PROGRAM Main
VAR
	// JaWa
	_iDbg:INT;	
	_download5:BOOL;
	//Enum1: FanControlTypes := FanControlTypes.Flow;
	GreenMaster: GreenMasterXXL_FB;
	StartupDone: BOOL;
	EventLog: EventLog;
	xxx: bool;
	Saver: FB_S_UPS_CX81xx;
	HostName: FB_GetHostName;
	UseReverse_C_QN1: BOOL;
	test1: bool;
	
	Std_Interface : Standard_Interface;
	CTH_Interface: CTH_Interface;
	Stena_Interface: Stena_Interface;
	ExtraAlarms_Interface: ExtraAlarms_Interface;
	SmokeControl_Interface: SmokeControl_Interface;

	Redundancy:Redundancy;
	ParallelUnits: ParallelUnits;
	
	GreenMasterDI: GreenMasterDI;
	GreenMasterDO: GreenMasterDO;
	GreenMasterAI: GreenMasterAI;
	GreenMasterAO: GreenMasterAO;
	GreenMasterAI2_RTU: GreenMasterAIU_ModbusRTU;
	AnySensorError: BOOL;
	{attribute 'TcEncoding':='UTF-8'}
	str: STRING;
	n: INT;
	
	NightCooling: BOOL;
	DebugStop: BOOL;
	WritePersistentData: WritePersistentData;
	StartWritePersistentData: BOOL;
	SavedParameters: GreenMasterBaseParameters;
	DevMon: DeviationMonitor;
	DevValue: LREAL;
	TestPID: TestPID;
	fbTime : FB_LocalSystemTime := ( bEnable := TRUE, dwCycle := 1 );
	LastSecondsCounter: LINT;
    sTime: STRING;	
	sPart1: STRING;
	sPart2: STRING;
	ExceptionYet: BOOL;
	PTest: POINTER TO BYTE;
	Crash: BOOL;
	i: INT;
	w: WORD;
	Rr: LREAL;
END_VAR
VAR PERSISTENT
END_VAR

IF NOT ExceptionYet THEN
	__TRY
		EventLog(EventLogData := Globals.EventLog);
		IF NOT StartupDone THEN
			Globals.SystemStartTime := NowDT();
			EventLog.LogEvent(Message := 'Starting up', Kind := EventTypes.Information);
			//EventLog.LogEventJSON(Message := 'Test data $${KFactor} and $${PressureControl.SP}', Kind := EventTypes.Debug, VarAdr := ADR(GreenMaster.Parameters.Regulation.ExtractAir), VarSize := SIZEOF(GreenMaster.Parameters.Regulation.ExtractAir), VarType := 'AirParameters');	
			StartupDone := TRUE;
		END_IF
		SavedParameters := GreenMaster.GetParameters();
		Globals.SystemUpTime := DT_TO_DWORD(NowDT()) - DT_TO_DWORD(Globals.SystemStartTime);
		
		NightCooling := FALSE;
		
		TestPID();
		
		str := '';
		FOR n := 0 TO GlobalSettings.MAX_COMPONENTS DO
			IF GlobalSettings.Components[n].Name = ComponentNames.NONE THEN
				EXIT;
			END_IF
			IF GlobalSettings.Components[n].EN THEN
				IF str <> '' THEN
					str := concat(str, ', ');
				END_IF
				str := concat(str, TO_STRING(GlobalSettings.Components[n].Name));
			END_IF
		END_FOR
		Globals.Components := str;
		
		HostName(bExecute := TRUE);
		// CX-503E98 CTH 1
		// CX-492F8F Diginet lab
		// CX-4F1CE6 NIBE AirSite lab
		// 
		Globals.HostName := HostName.sHostName; 
		IF F_ToUCase(HostName.sHostName) = 'CX-503E98' THEN
			UseReverse_C_QN1 := FALSE;
		ELSE
			UseReverse_C_QN1 := GreenMaster.Parameters.Io.AOutCalibration.C_QN1.InvertedOutput;
		END_IF
		
		IF GreenMaster.Parameters.System.Operation.IoUpdateEN THEN
			GreenMasterDI(DIn := Globals.IO.DIn, DInLevels := GreenMaster.Parameters.IO.DInLevels);
			GreenMasterDO(DOut := Globals.IO.DOut);
			GreenMasterAI(AIn := Globals.IO.AIn);
			GreenMasterAO(AOut := Globals.IO.AOut);
			GreenMasterAI2_RTU(Parameters:=GreenMaster.GetParameters(), EN:= TRUE);
		END_IF
		
		//_iDbg:=ComponentNames.GM_OPT_STENA;
		//Std_Interface(EN := GetComponent(Name := ComponentNames.GM_TAGS).EN, AIn := Globals.IO.AIn);
		Std_Interface(EN := GetComponent(Name := ComponentNames.GM_OPT_STD).EN, AIn := Globals.IO.AIn);
		CTH_Interface(EN := GetComponent(Name := ComponentNames.GM_OPT_CTH).EN, AIn := Globals.IO.AIn);	
		Stena_Interface(EN := GetComponent(Name := ComponentNames.GM_OPT_STENA).EN, AIn := Globals.IO.AIn);	
		
		// Redundant drift
		IF GetComponent(Name := ComponentNames.REDUNDANCY).EN THEN
			Redundancy(	EN := GetComponent(Name := ComponentNames.REDUNDANCY).EN,
						_UPPSTART_DONE:=StartupDone,
						_TF_CMD:=GreenMaster.Parameters.Regulation.SupplyAir.Control.CV > 0,
						_TF_V:=GreenMaster.Parameters.Regulation.SupplyAir.Control.CV > 0 AND GreenMaster.GetCurrentSupplyAirPV() > 10,
						_TF_OP:=LREAL_TO_REAL(GreenMaster.Parameters.Regulation.SupplyAir.Control.CV),
						_TL_GP_PV:=LREAL_TO_REAL(GreenMaster.GetCurrentSupplyAirPV()),
						_FF_CMD:=GreenMaster.Parameters.Regulation.ExtractAir.Control.CV > 0,
						_FF_V:=GreenMaster.Parameters.Regulation.ExtractAir.Control.CV > 0 AND GreenMaster.GetCurrentExtractAirPV() > 10,
						_FF_OP:=LREAL_TO_REAL(GreenMaster.Parameters.Regulation.ExtractAir.Control.CV),
						_FL_GP_PV:=LREAL_TO_REAL(GreenMaster.GetCurrentExtractAirPV()),
						_SERVICEBRYTARE:=FALSE
						);
		END_IF
		// Parallel units
		IF GetComponent(Name := ComponentNames.PARALLEL_UNITS).EN THEN
			ParallelUnits(	EN := GetComponent(Name := ComponentNames.PARALLEL_UNITS).EN,
							Tags := ADS_ParallelUnits.Tags,
							Parameters := GreenMaster.Parameters 
						);
		END_IF
		
		IF GetComponent(Name := ComponentNames.GM_OPT_CTH).EN THEN
			Globals.IO.DOut.DO15 := GreenMaster.Parameters.Alarm.Active.A.FireExtract;
			IF GreenMaster.Parameters.System.Operation.RemoteEN THEN
				IF GreenMaster.Parameters.IO.AIn.T_BT1 > (GreenMaster.Parameters.Regulation.NightCoolingLimit + 0.5) THEN
					NightCooling := CTH_Interface.NightCooling;	
				END_IF
				IF GreenMaster.Parameters.IO.AIn.T_BT1 < GreenMaster.Parameters.Regulation.NightCoolingLimit THEN
					NightCooling := FALSE;		
				END_IF
				GreenMaster.GetParameters().System.Operation.FireDamperUsed := FALSE;		
			END_IF
		END_IF
		
		IF GetComponent(Name := ComponentNames.GM_BASE).EN THEN
			GreenMaster.Update(DO_ := GreenMasterDO, AO := GreenMasterAO);
			GreenMaster(
				EN := TRUE AND (NOT DebugStop),
				RemoteEN := GreenMaster.Parameters.System.Operation.RemoteEN, //Std_Interface.ENO OR CTH_Interface.ENO OR Stena_Interface.ENO,	// TODO: Varför bara CTH här i original?  
				DI := GreenMasterDI,
				AI := GreenMasterAI,
				AI2 := GreenMasterAI2_RTU,
				TCP_AI := SmokeControl.GreenMasterSmokeControl,  
				Reverse_C_QN1 := UseReverse_C_QN1,
				NightCooling := NightCooling,
				EnableFansAndDampers := Std_Interface.EN OR Stena_Interface.EN OR (CTH_Interface.EN AND NOT CTH_Interface.FirePanelActive)
			);
		END_IF
		
		IF GetComponent(Name := ComponentNames.SIMULATION).EN THEN
			IF GreenMaster.GetParameters().System.Operation.Simulation THEN
				GreenMaster.Simulation(Parameters := GreenMaster.GetParameters(), Simulation := GreenMaster.GetParameters().Simulation);			
			END_IF
		END_IF
		
		AnySensorError := GreenMaster.Parameters.IO.AIn.F_BT1_Error OR 
			GreenMaster.Parameters.IO.AIn.T_BT2_Error OR
			GreenMaster.Parameters.IO.AIn.T_BT3_Error OR
			GreenMaster.Parameters.IO.AIn.H_BT1_Error OR
			GreenMaster.Parameters.IO.AIn.T_BT1_Error OR
			GreenMaster.Parameters.IO.AIn.BT1_Error OR
			GreenMaster.Parameters.IO.AIn.BT2_Error OR
			GreenMaster.Parameters.IO.AIn.F_BT2_Error OR	
			GreenMaster.Parameters.IO.AIn.F_BP1_Error OR
			GreenMaster.Parameters.IO.AIn.T_BP1_Error OR
			GreenMaster.Parameters.IO.AIn.F_BP2_Error OR
			GreenMaster.Parameters.IO.AIn.T_BP2_Error OR
			GreenMaster.Parameters.IO.AIn.F_BP3_Error OR
			GreenMaster.Parameters.IO.AIn.T_BF1_Error OR
			GreenMaster.Parameters.IO.AIn.F_BF1_Error;	
		
		
		// Save persistent data on power off or fail
		Saver();
		WritePersistentData(NETID := '', PORT := 851, TMOUT := T#10S, START := StartWritePersistentData);
		
		DevMon(Value := DevValue, TargetValue := 5);
		
		IF GetComponent(Name := ComponentNames.EXTRA_ALARMS).EN THEN	
			GreenMaster.GetParameters().Alarm.Status.A.AL01 := NOT ExtraAlarmInputs.AL01;
			GreenMaster.GetParameters().Alarm.Status.A.AL02 := NOT ExtraAlarmInputs.AL02;
			GreenMaster.GetParameters().Alarm.Status.A.AL03 := NOT ExtraAlarmInputs.AL03;
			GreenMaster.GetParameters().Alarm.Status.A.AL04 := NOT ExtraAlarmInputs.AL04;
			GreenMaster.GetParameters().Alarm.Status.A.AL05 := NOT ExtraAlarmInputs.AL05;
			GreenMaster.GetParameters().Alarm.Status.A.AL06 := NOT ExtraAlarmInputs.AL06;
			GreenMaster.GetParameters().Alarm.Status.A.AL07 := NOT ExtraAlarmInputs.AL07;
			GreenMaster.GetParameters().Alarm.Status.A.AL08 := NOT ExtraAlarmInputs.AL08;
		END_IF
		ExtraAlarms_Interface(EN := GetComponent(Name := ComponentNames.EXTRA_ALARMS).EN);
		SmokeControl_Interface(EN := GetComponent(Name := ComponentNames.GM_SMOKE_CONTROL).EN);
		fbtime();
		IF Globals.SecondsCounter <> LastSecondsCounter THEN
			LastSecondsCounter := Globals.SecondsCounter;
			// 2021-11-10-08:08:53.582
			sTime := SYSTEMTIME_TO_STRING(fbTime.systemTime);
			sPart1 := Delete(sTime, 4, 19);
			sPart2 := Replace(sPart1, ' ', 1, 11);
			GreenMaster.GetParameters().System.SystemTime := sPart2;
		END_IF
		IF Crash THEN
			PTest^ := 111;
		END_IF
	__CATCH
		ExceptionYet := TRUE; 			
	__ENDTRY
ELSE
	ExceptionYet := TRUE; 	
END_IF

Rr := -4;
i := TO_INT(Rr);
i := TO_INT(w);

END_PROGRAM

(* stored: Version 1.1.0.1, ProductVersion 3.1.4024.6
   POU Main: Id {0fc71ecf-56d1-4789-9140-ae6c41febaf6}, SpecialFunc None *)
